ABB RobotStudio station: solution.rsstn

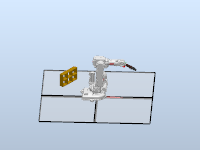
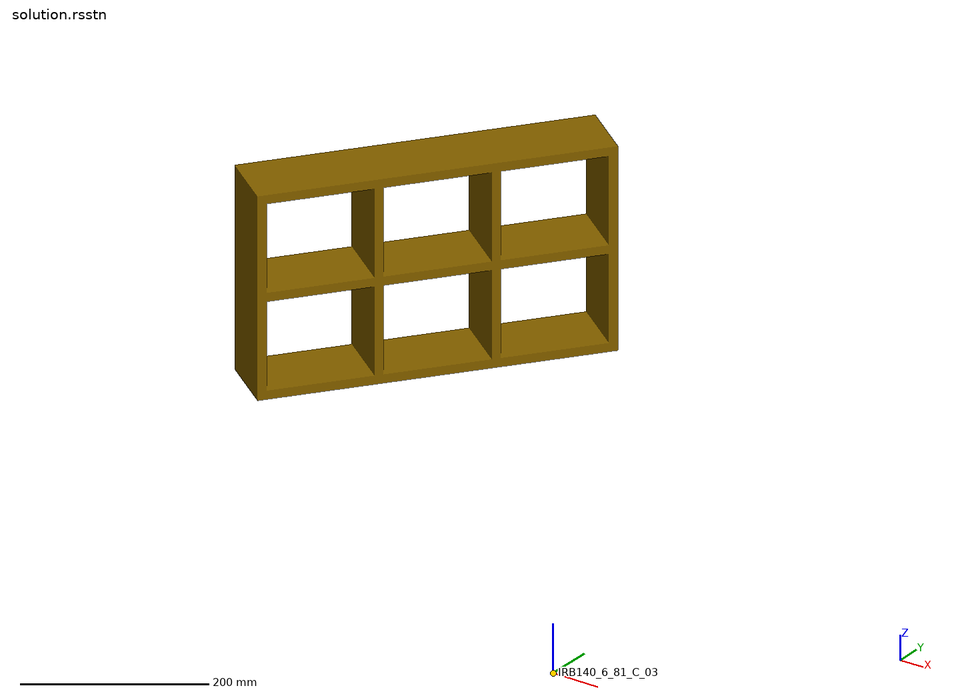
[picture v1: parts stored in the station drawn from their meshes, with robot base, taught points and paths (robot models come from the ABB library and are not in the file)]
Station solution (saved by RobotStudio 22.1.9826.0)
Controller IRB140_6_81
  mechanical unit ROB_1: IRB140_6_81_C_03, 6 joints, base frame (0, 0, 0) mm
Layout (positions relative to the parent item):
  - IRB140_6_81_C_03 [mechanism, from Robots\IRB140_6_81_C_G_03.rslib] at (0, 0, 0) mm; joint values [0, 0, 0, 0, 0.5236, 0] (rad or m)
  - stand [part] at (-573.19, 563.59, 121.97) mm, rotated rx 0 ry 90 rz -37.36 deg, size 240 x 400 x 80 mm
  - gripper [mechanism, from libs\gripper.rslib] at (506.29, 0, 679.5) mm, rotated rx 180 ry 60 rz 180 deg
